(* Logix 5000 project; controller PRU vendor 1 type 14 code 107 rev 20.13; software revision 20.01; part 2 of 17 *)
(* tags used below, declared in another part *)
   RIGHT_ENCODER_DEG_OUT_REAL_OUT : REAL;
   LEFT_ENCODER_DEG_WAS_SCANRATE_MOVED_OUT : REAL;
   RIGHT_ENCODER_DEG_WAS_SCANRATE_MOVED_OUT : REAL;
   MASTER_RIGHT_BOOL_IN : BOOL;
   ENCODER_MOVED_LAST_SEC_REAL_OUT : REAL;
   MIX_REV_PER_MIN_REAL_OUT : REAL;
   RETENTION_TIME_MIN_REAL_OUT : REAL;
   MIX_FWD_PRESET_REAL_IN : REAL;
   MIX_REV_PRESET_REAL_IN : REAL;
   AUTO_FWD_CMD_BOOL_OUT : BOOL;
   ENCODER_ACC_REAL_OUT : REAL;
   SREW_MODE_INT_IN : INT;
   SCREW_PITCH_CONSTANT_REAL_IN : REAL;
   MIX_SEQ : INT;
   ONE_SECOND_ENCODER_SCAN : BOOL;   // 100 x 10mS.
   RIGHT_ENCODER_DEG_WAS_SCANRATE : REAL;
   MIX_SEQ_STEP_00_DONE_TON : TIMER;
   MIX_SEQ_STEP_01_DONE : BOOL;
   MIX_SEQ_STEP_02_DONE : BOOL;
   MIX_STEP_00_ION : BOOL;
   MIX_STEP_01_ION : BOOL;   // FORWARD
   MIX_STEP_01_ONSN : BOOL;
   MIX_STEP_01_ONSP : BOOL;
   MIX_FWD_SS : BOOL;
   MIX_CYC_TIME_ACC : DINT;
   MIX_CYC_TIME : REAL;
   MIX_FWD_DEG : REAL;
   MIX_DEG_PER_SEC : REAL;
   MIX_STEP_02_ION : BOOL;   // REVERSE
   FWD_CMD_BON : TIMER;
   REV_CMD_BON : TIMER;
   Revision : DINT;
   SCREW_ENCODERS : SCREW_ENCODERS;
   SCREW_SPEED : SCREW_SPEED;
(* SCREW_ENCODERS, continued *)

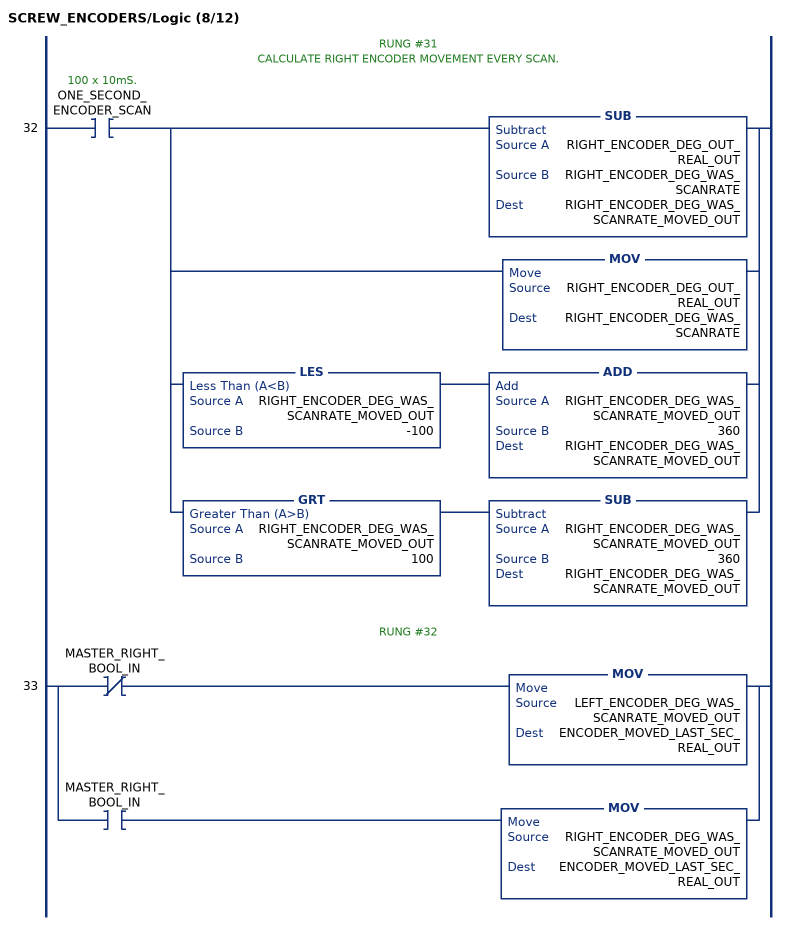
   // RUNG #31
   // CALCULATE RIGHT ENCODER MOVEMENT EVERY SCAN.
   32: XIC(ONE_SECOND_ENCODER_SCAN)[SUB(RIGHT_ENCODER_DEG_OUT_REAL_OUT,RIGHT_ENCODER_DEG_WAS_SCANRATE,RIGHT_ENCODER_DEG_WAS_SCANRATE_MOVED_OUT) ,MOV(RIGHT_ENCODER_DEG_OUT_REAL_OUT,RIGHT_ENCODER_DEG_WAS_SCANRATE) ,LES(RIGHT_ENCODER_DEG_WAS_SCANRATE_MOVED_OUT,-100) ADD(RIGHT_ENCODER_DEG_WAS_SCANRATE_MOVED_OUT,360,RIGHT_ENCODER_DEG_WAS_SCANRATE_MOVED_OUT) ,GRT(RIGHT_ENCODER_DEG_WAS_SCANRATE_MOVED_OUT,100) SUB(RIGHT_ENCODER_DEG_WAS_SCANRATE_MOVED_OUT,360,RIGHT_ENCODER_DEG_WAS_SCANRATE_MOVED_OUT) ];
   // RUNG #32
   33: [XIO(MASTER_RIGHT_BOOL_IN) MOV(LEFT_ENCODER_DEG_WAS_SCANRATE_MOVED_OUT,ENCODER_MOVED_LAST_SEC_REAL_OUT) ,XIC(MASTER_RIGHT_BOOL_IN) MOV(RIGHT_ENCODER_DEG_WAS_SCANRATE_MOVED_OUT,ENCODER_MOVED_LAST_SEC_REAL_OUT) ];
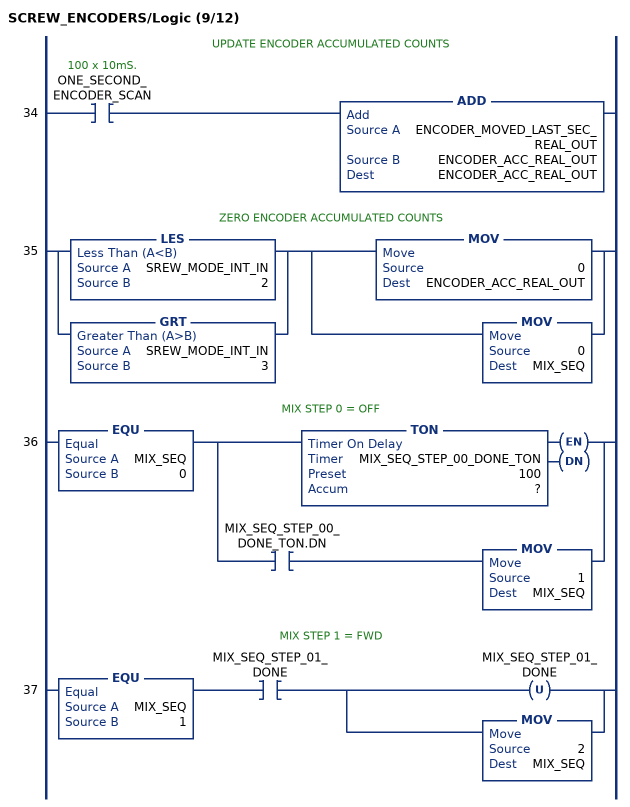
   // UPDATE ENCODER ACCUMULATED COUNTS
   34: XIC(ONE_SECOND_ENCODER_SCAN)ADD(ENCODER_MOVED_LAST_SEC_REAL_OUT,ENCODER_ACC_REAL_OUT,ENCODER_ACC_REAL_OUT);
   // ZERO ENCODER ACCUMULATED COUNTS
   35: [LES(SREW_MODE_INT_IN,2) ,GRT(SREW_MODE_INT_IN,3) ][MOV(0,ENCODER_ACC_REAL_OUT) ,MOV(0,MIX_SEQ) ];
   // MIX STEP 0 = OFF
   36: EQU(MIX_SEQ,0)[TON(MIX_SEQ_STEP_00_DONE_TON,?,?) ,XIC(MIX_SEQ_STEP_00_DONE_TON.DN) MOV(1,MIX_SEQ) ];
   // MIX STEP 1 = FWD
   37: EQU(MIX_SEQ,1)XIC(MIX_SEQ_STEP_01_DONE)[OTU(MIX_SEQ_STEP_01_DONE) ,MOV(2,MIX_SEQ) ];
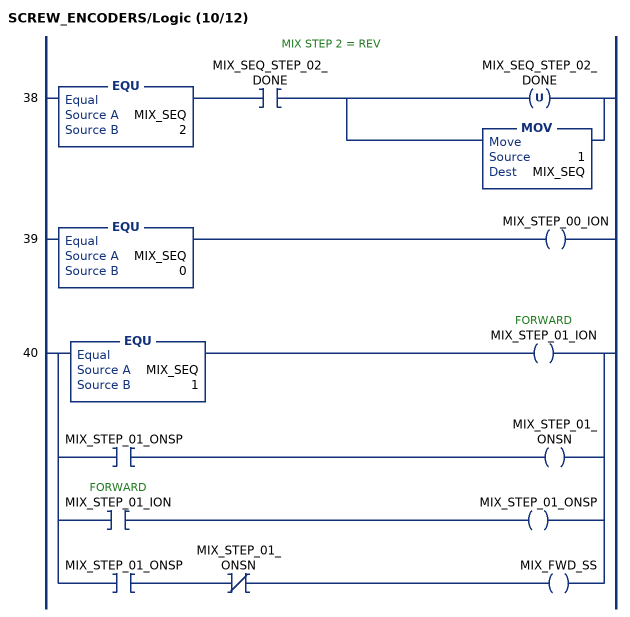
   // MIX STEP 2 = REV
   38: EQU(MIX_SEQ,2)XIC(MIX_SEQ_STEP_02_DONE)[OTU(MIX_SEQ_STEP_02_DONE) ,MOV(1,MIX_SEQ) ];
   39: EQU(MIX_SEQ,0)OTE(MIX_STEP_00_ION);
   40: [EQU(MIX_SEQ,1) OTE(MIX_STEP_01_ION) ,XIC(MIX_STEP_01_ONSP) OTE(MIX_STEP_01_ONSN) ,XIC(MIX_STEP_01_ION) OTE(MIX_STEP_01_ONSP) ,XIC(MIX_STEP_01_ONSP) XIO(MIX_STEP_01_ONSN) OTE(MIX_FWD_SS) ];
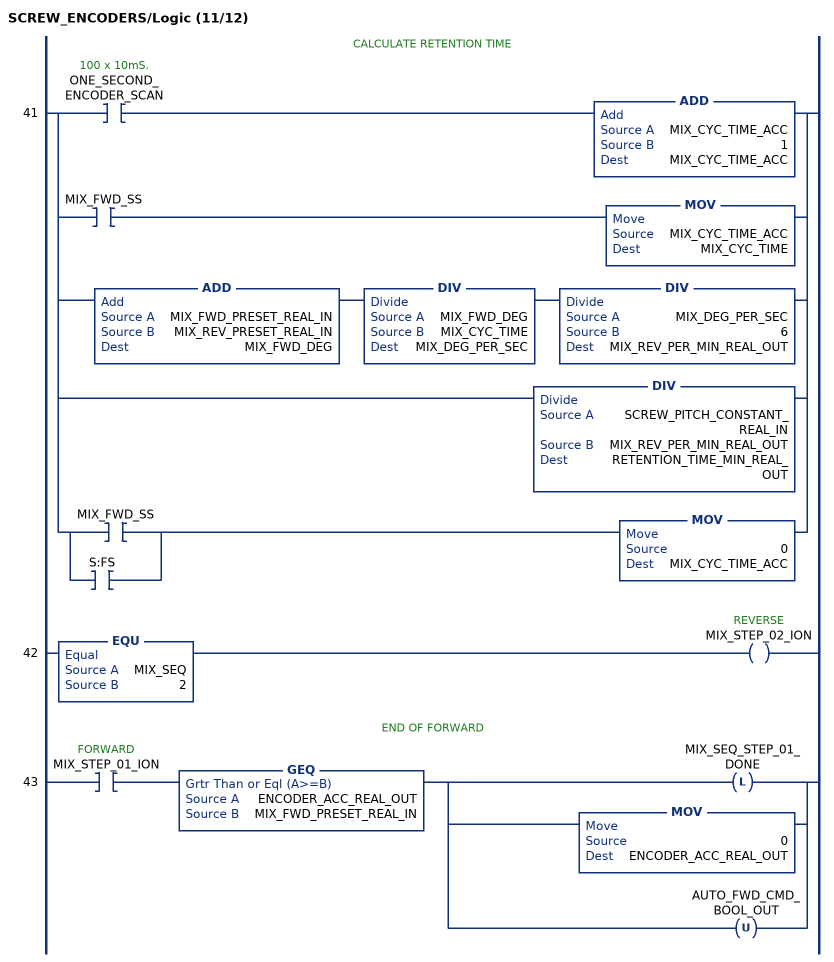
   // CALCULATE RETENTION TIME
   41: [XIC(ONE_SECOND_ENCODER_SCAN) ADD(MIX_CYC_TIME_ACC,1,MIX_CYC_TIME_ACC) ,XIC(MIX_FWD_SS) MOV(MIX_CYC_TIME_ACC,MIX_CYC_TIME) ,ADD(MIX_FWD_PRESET_REAL_IN,MIX_REV_PRESET_REAL_IN,MIX_FWD_DEG) DIV(MIX_FWD_DEG,MIX_CYC_TIME,MIX_DEG_PER_SEC) DIV(MIX_DEG_PER_SEC,6,MIX_REV_PER_MIN_REAL_OUT) ,DIV(SCREW_PITCH_CONSTANT_REAL_IN,MIX_REV_PER_MIN_REAL_OUT,RETENTION_TIME_MIN_REAL_OUT) ,[XIC(MIX_FWD_SS) ,XIC(S:FS) ] MOV(0,MIX_CYC_TIME_ACC) ];
   42: EQU(MIX_SEQ,2)OTE(MIX_STEP_02_ION);
   // END OF FORWARD
   43: XIC(MIX_STEP_01_ION)GEQ(ENCODER_ACC_REAL_OUT,MIX_FWD_PRESET_REAL_IN)[OTL(MIX_SEQ_STEP_01_DONE) ,MOV(0,ENCODER_ACC_REAL_OUT) ,OTU(AUTO_FWD_CMD_BOOL_OUT) ];
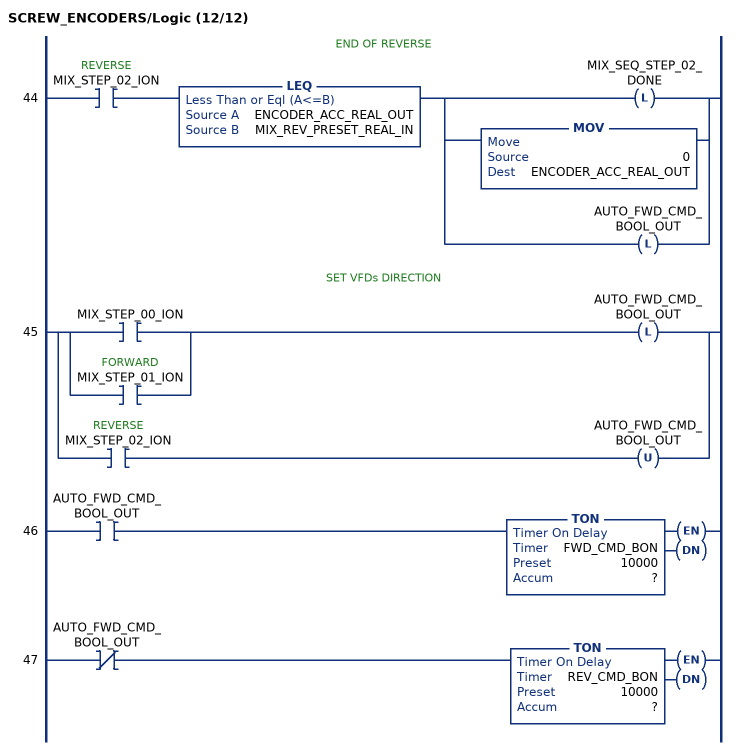
   // END OF REVERSE
   44: XIC(MIX_STEP_02_ION)LEQ(ENCODER_ACC_REAL_OUT,MIX_REV_PRESET_REAL_IN)[OTL(MIX_SEQ_STEP_02_DONE) ,MOV(0,ENCODER_ACC_REAL_OUT) ,OTL(AUTO_FWD_CMD_BOOL_OUT) ];
   // SET VFDs DIRECTION
   45: [[XIC(MIX_STEP_00_ION) ,XIC(MIX_STEP_01_ION) ] OTL(AUTO_FWD_CMD_BOOL_OUT) ,XIC(MIX_STEP_02_ION) OTU(AUTO_FWD_CMD_BOOL_OUT) ];
   46: XIC(AUTO_FWD_CMD_BOOL_OUT)TON(FWD_CMD_BON,?,?);
   47: XIO(AUTO_FWD_CMD_BOOL_OUT)TON(REV_CMD_BON,?,?);
END_ROUTINE
END_ADD_ON_INSTRUCTION

ADD_ON_INSTRUCTION SCREW_SPEED   (* revision 1.0, vendor Deterministic Systems, Inc. *)
VAR_INPUT
   IN_SCREW_MODE : INT; {required}
   IN_AUTO_FWD_CMD_BOOL : BOOL; {required}
   IN_MASTER_RIGHT_BOOL : BOOL; {required}
   IN_VFD_STOP_CMD : BOOL; {required}
   IN_DCS_AUTO_SCREW_CMD_PCNT : REAL; {required}
END_VAR
VAR_OUTPUT
   OUT_DCS_MASTER_SPEED_CMD : REAL; {access Read Only, required}
END_VAR
VAR_INPUT
   IN_HMI_SEMIAUTO_SCREW_CMD_PCNT : REAL; {required}
END_VAR
VAR_OUTPUT
   OUT_MASTER_AUTO_SETPOINT_PCNT : REAL; {access Read Only, required}
END_VAR
VAR_INPUT
   IN_LEFT_RIGHT_ENCODER_ERROR_DEG : REAL; {required}
   IN_WIPER_OSC_SETPOINT : REAL; {required}
END_VAR
VAR_OUTPUT
   OUT_FINAL_SCREW_POSITION_ERROR : REAL; {access Read Only, required}
   OUT_AUTO_SCREW_LEFT_CMD_FREQ : REAL; {access Read Only, required}
   OUT_AUTO_SCREW_RIGHT_CMD_FREQ : REAL; {access Read Only, required}
END_VAR
VAR_INPUT
   IN_LEFT_VFD_ION : BOOL; {required}
   IN_RIGHT_VFD_ION : BOOL; {required}
   IN_LEFT_VFD_ACTUAL : BOOL; {required}
   IN_RIGHT_VFD_ACTUAL : BOOL; {required}
END_VAR
VAR_OUTPUT
   OUT_FORCE_ZERO_SPEED : BOOL; {access Read Only, required}
END_VAR
VAR_INPUT
   IN_SCREW_FAULTED_IOK : BOOL; {required}
END_VAR
VAR_OUTPUT
   OUT_LEFT_AUTO_PCNT_SETPOINT : REAL; {access Read Only, required}
   OUT_RIGHT_AUTO_PCNT_SETPOINT : REAL; {access Read Only, required}
END_VAR
VAR_INPUT
   IN_LEFT_VFD_ACTUAL_FREQ : INT; {required}
   IN_RIGHT_VFD_ACTUAL_FREQ : INT; {required}
END_VAR
VAR_OUTPUT
   OUT_LEFT_VFD_ACTUAL_SPEED_PERCENT : REAL; {required}
   OUT_RIGHT_VFD_ACTUAL_SPEED_PERCENT : REAL; {access Read Only, required}
   CALC_COMP_LIMIT : REAL; {access None, required}
END_VAR
VAR_INPUT
   IN_SET_ZERO_SPEED : BOOL; {required}
END_VAR
VAR
   SCREW_MODE_AUTO : BOOL;
   DCS_MASTER_SPEED_CMD : REAL;
   SLAVE_COMPENSATION_GAIN : REAL;
   SLAVE_COMPENSATION_PER_DEGREE : REAL;
   SLAVE_AUTO_SETPOINT_PCNT : REAL;
   RIGHT_MAX_COMP_PCNT : REAL;
   RIGHT_MIN_COMP_PCNT : REAL;
   RPM_FREQ_MULTIPLIER : REAL := 711.16;
   MASTER_SETPOINT_END : REAL; {access None}
   CALC_MASTER_SETPOINT : REAL; {access None}
   ROC : DSi_COMP_SCALE; {access None}
   FWD_MASTER_AUTO_SETPOINT_PCNT : REAL; {access None}
   CALC_COMP_LIMIT_REV : REAL; {access None}
   REV_MASTER_AUTO_SETPOINT_PCNT : REAL; {access None}
   MASTER_SETPOINT_END_REV : REAL; {access None}
   ROC2 : DSi_COMP_SCALE; {access None}
END_VAR

ROUTINE Logic   (* ladder *)
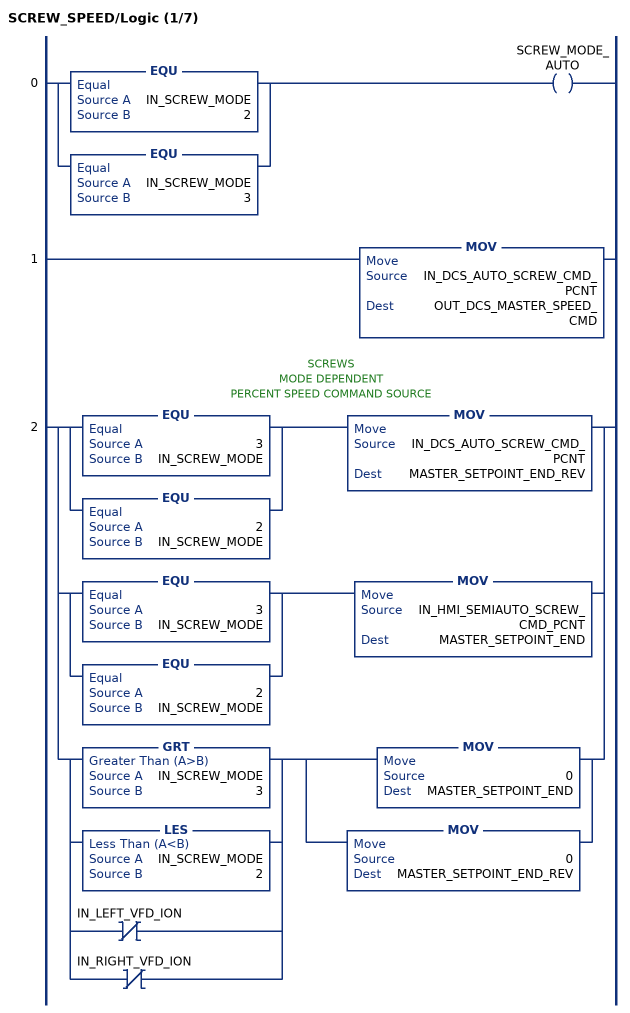
   0: [EQU(IN_SCREW_MODE,2) ,EQU(IN_SCREW_MODE,3) ]OTE(SCREW_MODE_AUTO);
   1: MOV(IN_DCS_AUTO_SCREW_CMD_PCNT,OUT_DCS_MASTER_SPEED_CMD);
   // SCREWS
   // MODE DEPENDENT
   // PERCENT SPEED COMMAND SOURCE
   2: [[EQU(3,IN_SCREW_MODE) ,EQU(2,IN_SCREW_MODE) ] MOV(IN_DCS_AUTO_SCREW_CMD_PCNT,MASTER_SETPOINT_END_REV) ,[EQU(3,IN_SCREW_MODE) ,EQU(2,IN_SCREW_MODE) ] MOV(IN_HMI_SEMIAUTO_SCREW_CMD_PCNT,MASTER_SETPOINT_END) ,[GRT(IN_SCREW_MODE,3) ,LES(IN_SCREW_MODE,2) ,XIO(IN_LEFT_VFD_ION) ,XIO(IN_RIGHT_VFD_ION) ] [MOV(0,MASTER_SETPOINT_END) ,MOV(0,MASTER_SETPOINT_END_REV) ] ];
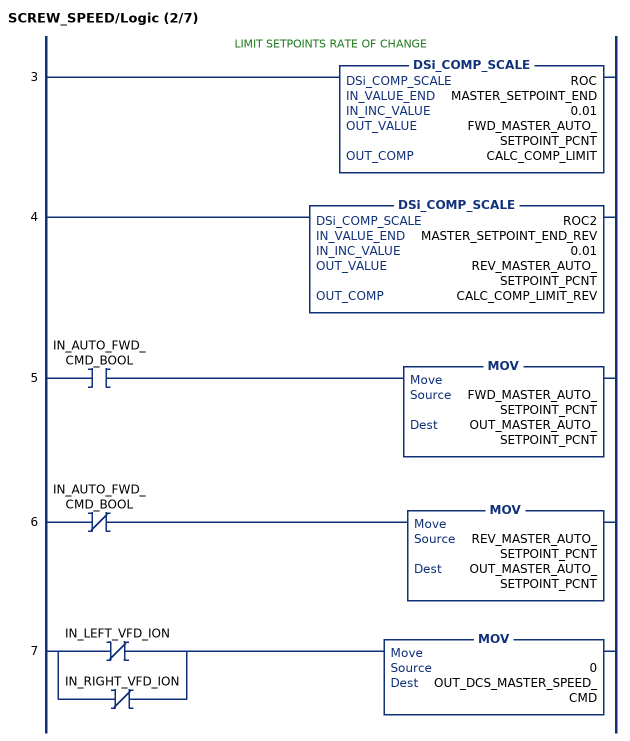
   // LIMIT SETPOINTS RATE OF CHANGE
   3: DSi_COMP_SCALE(ROC,MASTER_SETPOINT_END,0.01,FWD_MASTER_AUTO_SETPOINT_PCNT,CALC_COMP_LIMIT);
   4: DSi_COMP_SCALE(ROC2,MASTER_SETPOINT_END_REV,0.01,REV_MASTER_AUTO_SETPOINT_PCNT,CALC_COMP_LIMIT_REV);
   5: XIC(IN_AUTO_FWD_CMD_BOOL)MOV(FWD_MASTER_AUTO_SETPOINT_PCNT,OUT_MASTER_AUTO_SETPOINT_PCNT);
   6: XIO(IN_AUTO_FWD_CMD_BOOL)MOV(REV_MASTER_AUTO_SETPOINT_PCNT,OUT_MASTER_AUTO_SETPOINT_PCNT);
   7: [XIO(IN_LEFT_VFD_ION) ,XIO(IN_RIGHT_VFD_ION) ]MOV(0,OUT_DCS_MASTER_SPEED_CMD);
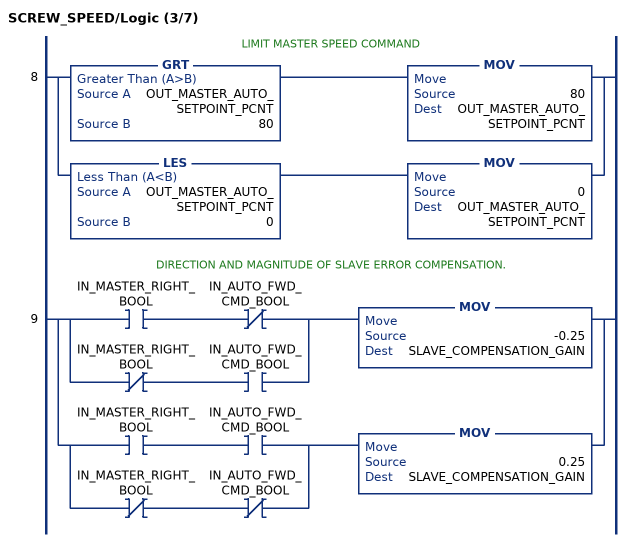
   // LIMIT MASTER SPEED COMMAND
   8: [GRT(OUT_MASTER_AUTO_SETPOINT_PCNT,80) MOV(80,OUT_MASTER_AUTO_SETPOINT_PCNT) ,LES(OUT_MASTER_AUTO_SETPOINT_PCNT,0) MOV(0,OUT_MASTER_AUTO_SETPOINT_PCNT) ];
   // DIRECTION AND MAGNITUDE OF SLAVE ERROR COMPENSATION.
   9: [[XIC(IN_MASTER_RIGHT_BOOL) XIO(IN_AUTO_FWD_CMD_BOOL) ,XIO(IN_MASTER_RIGHT_BOOL) XIC(IN_AUTO_FWD_CMD_BOOL) ] MOV(-0.25,SLAVE_COMPENSATION_GAIN) ,[XIC(IN_MASTER_RIGHT_BOOL) XIC(IN_AUTO_FWD_CMD_BOOL) ,XIO(IN_MASTER_RIGHT_BOOL) XIO(IN_AUTO_FWD_CMD_BOOL) ] MOV(0.25,SLAVE_COMPENSATION_GAIN) ];
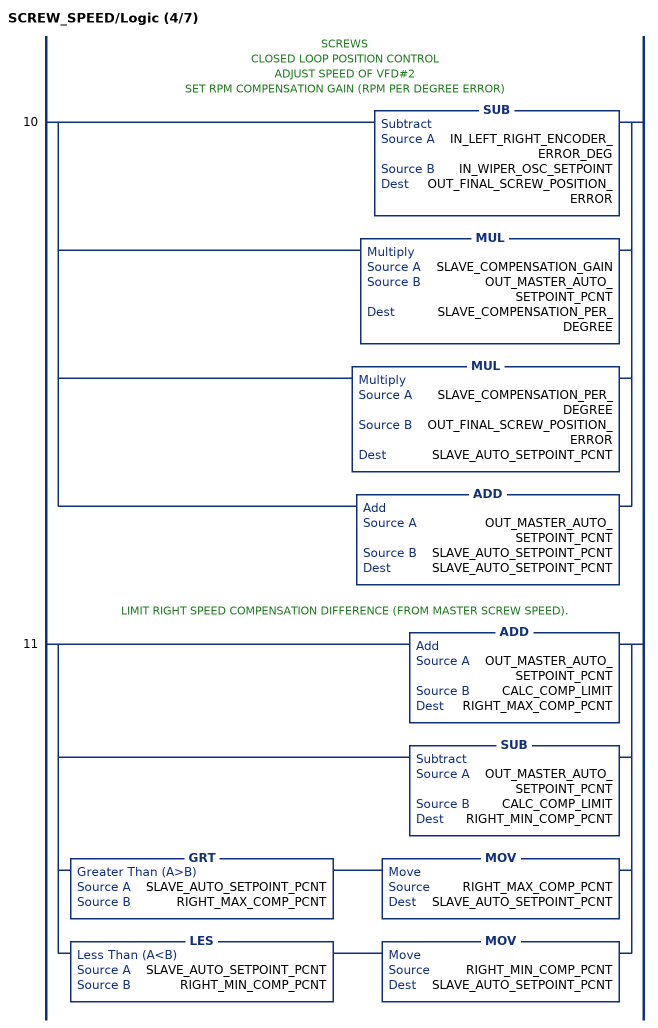
   // SCREWS
   // CLOSED LOOP POSITION CONTROL
   // ADJUST SPEED OF VFD#2
   // SET RPM COMPENSATION GAIN (RPM PER DEGREE ERROR)
   10: [SUB(IN_LEFT_RIGHT_ENCODER_ERROR_DEG,IN_WIPER_OSC_SETPOINT,OUT_FINAL_SCREW_POSITION_ERROR) ,MUL(SLAVE_COMPENSATION_GAIN,OUT_MASTER_AUTO_SETPOINT_PCNT,SLAVE_COMPENSATION_PER_DEGREE) ,MUL(SLAVE_COMPENSATION_PER_DEGREE,OUT_FINAL_SCREW_POSITION_ERROR,SLAVE_AUTO_SETPOINT_PCNT) ,ADD(OUT_MASTER_AUTO_SETPOINT_PCNT,SLAVE_AUTO_SETPOINT_PCNT,SLAVE_AUTO_SETPOINT_PCNT) ];
   // LIMIT RIGHT SPEED COMPENSATION DIFFERENCE (FROM MASTER SCREW SPEED).
   11: [ADD(OUT_MASTER_AUTO_SETPOINT_PCNT,CALC_COMP_LIMIT,RIGHT_MAX_COMP_PCNT) ,SUB(OUT_MASTER_AUTO_SETPOINT_PCNT,CALC_COMP_LIMIT,RIGHT_MIN_COMP_PCNT) ,GRT(SLAVE_AUTO_SETPOINT_PCNT,RIGHT_MAX_COMP_PCNT) MOV(RIGHT_MAX_COMP_PCNT,SLAVE_AUTO_SETPOINT_PCNT) ,LES(SLAVE_AUTO_SETPOINT_PCNT,RIGHT_MIN_COMP_PCNT) MOV(RIGHT_MIN_COMP_PCNT,SLAVE_AUTO_SETPOINT_PCNT) ];
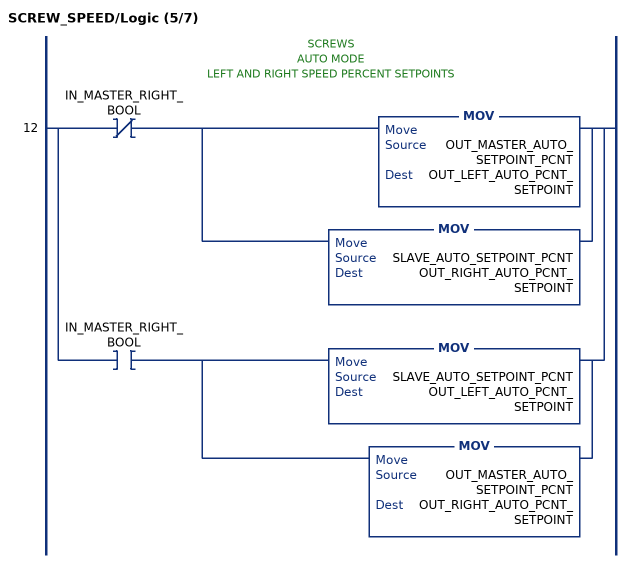
   // SCREWS
   // AUTO MODE
   // LEFT AND RIGHT SPEED PERCENT SETPOINTS
   12: [XIO(IN_MASTER_RIGHT_BOOL) [MOV(OUT_MASTER_AUTO_SETPOINT_PCNT,OUT_LEFT_AUTO_PCNT_SETPOINT) ,MOV(SLAVE_AUTO_SETPOINT_PCNT,OUT_RIGHT_AUTO_PCNT_SETPOINT) ] ,XIC(IN_MASTER_RIGHT_BOOL) [MOV(SLAVE_AUTO_SETPOINT_PCNT,OUT_LEFT_AUTO_PCNT_SETPOINT) ,MOV(OUT_MASTER_AUTO_SETPOINT_PCNT,OUT_RIGHT_AUTO_PCNT_SETPOINT) ] ];
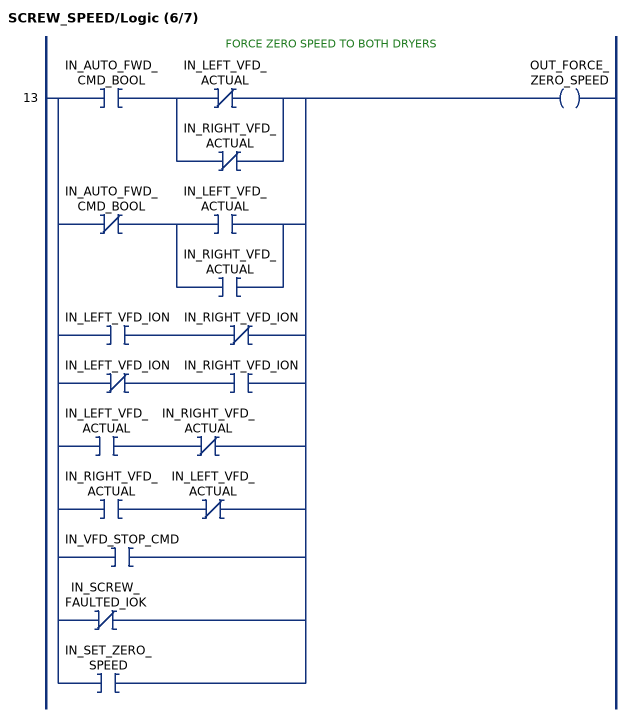
   // FORCE ZERO SPEED TO BOTH DRYERS
   13: [XIC(IN_AUTO_FWD_CMD_BOOL) [XIO(IN_LEFT_VFD_ACTUAL) ,XIO(IN_RIGHT_VFD_ACTUAL) ] ,XIO(IN_AUTO_FWD_CMD_BOOL) [XIC(IN_LEFT_VFD_ACTUAL) ,XIC(IN_RIGHT_VFD_ACTUAL) ] ,XIC(IN_LEFT_VFD_ION) XIO(IN_RIGHT_VFD_ION) ,XIO(IN_LEFT_VFD_ION) XIC(IN_RIGHT_VFD_ION) ,XIC(IN_LEFT_VFD_ACTUAL) XIO(IN_RIGHT_VFD_ACTUAL) ,XIC(IN_RIGHT_VFD_ACTUAL) XIO(IN_LEFT_VFD_ACTUAL) ,XIC(IN_VFD_STOP_CMD) ,XIO(IN_SCREW_FAULTED_IOK) ,XIC(IN_SET_ZERO_SPEED) ]OTE(OUT_FORCE_ZERO_SPEED);
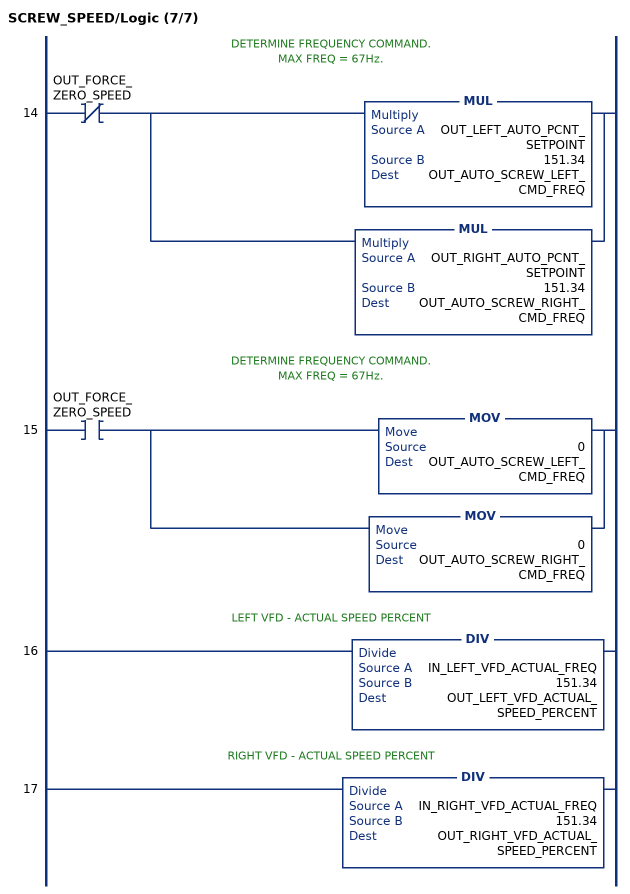
   // DETERMINE FREQUENCY COMMAND.
   // MAX FREQ = 67Hz.
   14: XIO(OUT_FORCE_ZERO_SPEED)[MUL(OUT_LEFT_AUTO_PCNT_SETPOINT,151.34,OUT_AUTO_SCREW_LEFT_CMD_FREQ) ,MUL(OUT_RIGHT_AUTO_PCNT_SETPOINT,151.34,OUT_AUTO_SCREW_RIGHT_CMD_FREQ) ];
   // DETERMINE FREQUENCY COMMAND.
   // MAX FREQ = 67Hz.
   15: XIC(OUT_FORCE_ZERO_SPEED)[MOV(0,OUT_AUTO_SCREW_LEFT_CMD_FREQ) ,MOV(0,OUT_AUTO_SCREW_RIGHT_CMD_FREQ) ];
   // LEFT VFD - ACTUAL SPEED PERCENT
   16: DIV(IN_LEFT_VFD_ACTUAL_FREQ,151.34,OUT_LEFT_VFD_ACTUAL_SPEED_PERCENT);
   // RIGHT VFD - ACTUAL SPEED PERCENT
   17: DIV(IN_RIGHT_VFD_ACTUAL_FREQ,151.34,OUT_RIGHT_VFD_ACTUAL_SPEED_PERCENT);
END_ROUTINE
END_ADD_ON_INSTRUCTION

ADD_ON_INSTRUCTION SCREW_WIPER   (* revision 1.0, vendor Deterministic Systems, Inc. *)
VAR_INPUT
   HMI_WIPE_INC_REAL_IN : REAL; {required}
   HMI_WIPE_SETPOINT_REAL_IN : REAL; {required}
   WIPE_HOLD_TIME_DINT_IN : DINT; {required}
END_VAR
VAR_OUTPUT
   WIPE_HOLDING_BOOL_OUT : BOOL; {access Read Only, required}
   WIPER_OSC_REAL_OUT : REAL; {access Read Only, required}
END_VAR
VAR_INPUT
   WIPE_EON_IN : BOOL; {required}
   WIPE_FREEZE_IN : BOOL; {required}
END_VAR
VAR
   SCREWS_TON : TIMER := (PRE := 10000);
   WIPE_INC : REAL;
   WIPE_PLUS_HOLD_VALUE : REAL;
   WIPE_MINUS_HOLD_VALUE : REAL;
   SCREWS_PLUS_HOLD_ONSN : BOOL;
   SCREWS_PLUS_HOLD_ONSP : BOOL;
   SCREWS_PLUS_HOLD_SS : BOOL;
   SCREWS_PLUS_HOLD : BOOL;
   SCREWS_MINUS_HOLD_ONSN : BOOL;
   SCREWS_MINUS_HOLD_ONSP : BOOL;
   SCREWS_MINUS_HOLD_SS : BOOL;
   SCREWS_MINUS_HOLD : BOOL;
   WIPE_HOLD_TIMER : TIMER := (PRE := 5000);
   WIPE_SIN_INDEX : REAL;
   WIPE_SINE : REAL;
   HMI_WIPE_SETPOINT_REAL : REAL; {access None}
   HMI_WIPE_SETPOINT_COMP : REAL; {access None}
   ROC_WIPE_SETPOINT : DSi_COMP_SCALE; {access None}
END_VAR

ROUTINE Logic   (* ladder *)
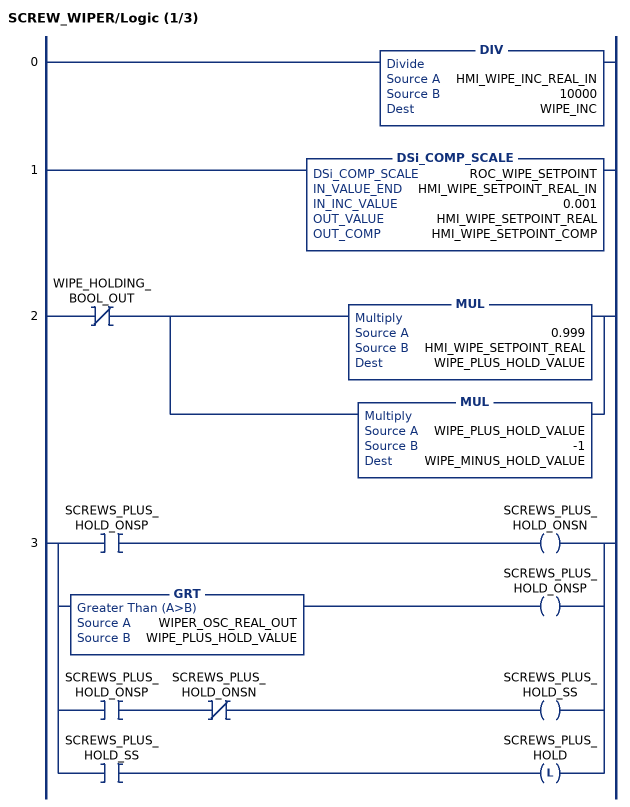
   0: DIV(HMI_WIPE_INC_REAL_IN,10000,WIPE_INC);
   1: DSi_COMP_SCALE(ROC_WIPE_SETPOINT,HMI_WIPE_SETPOINT_REAL_IN,0.001,HMI_WIPE_SETPOINT_REAL,HMI_WIPE_SETPOINT_COMP);
   2: XIO(WIPE_HOLDING_BOOL_OUT)[MUL(0.999,HMI_WIPE_SETPOINT_REAL,WIPE_PLUS_HOLD_VALUE) ,MUL(WIPE_PLUS_HOLD_VALUE,-1,WIPE_MINUS_HOLD_VALUE) ];
   3: [XIC(SCREWS_PLUS_HOLD_ONSP) OTE(SCREWS_PLUS_HOLD_ONSN) ,GRT(WIPER_OSC_REAL_OUT,WIPE_PLUS_HOLD_VALUE) OTE(SCREWS_PLUS_HOLD_ONSP) ,XIC(SCREWS_PLUS_HOLD_ONSP) XIO(SCREWS_PLUS_HOLD_ONSN) OTE(SCREWS_PLUS_HOLD_SS) ,XIC(SCREWS_PLUS_HOLD_SS) OTL(SCREWS_PLUS_HOLD) ];
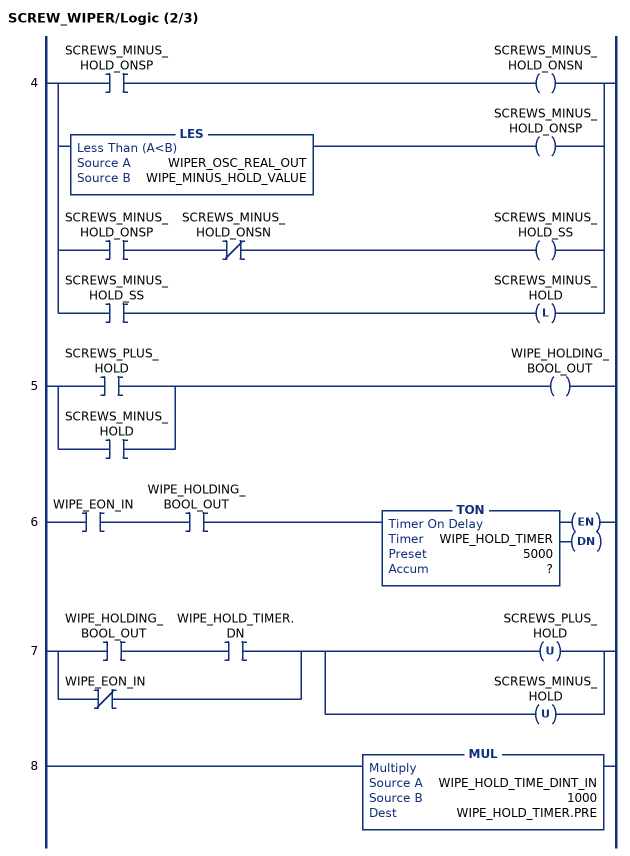
   4: [XIC(SCREWS_MINUS_HOLD_ONSP) OTE(SCREWS_MINUS_HOLD_ONSN) ,LES(WIPER_OSC_REAL_OUT,WIPE_MINUS_HOLD_VALUE) OTE(SCREWS_MINUS_HOLD_ONSP) ,XIC(SCREWS_MINUS_HOLD_ONSP) XIO(SCREWS_MINUS_HOLD_ONSN) OTE(SCREWS_MINUS_HOLD_SS) ,XIC(SCREWS_MINUS_HOLD_SS) OTL(SCREWS_MINUS_HOLD) ];
   5: [XIC(SCREWS_PLUS_HOLD) ,XIC(SCREWS_MINUS_HOLD) ]OTE(WIPE_HOLDING_BOOL_OUT);
   6: XIC(WIPE_EON_IN)XIC(WIPE_HOLDING_BOOL_OUT)TON(WIPE_HOLD_TIMER,?,?);
   7: [XIC(WIPE_HOLDING_BOOL_OUT) XIC(WIPE_HOLD_TIMER.DN) ,XIO(WIPE_EON_IN) ][OTU(SCREWS_PLUS_HOLD) ,OTU(SCREWS_MINUS_HOLD) ];
   8: MUL(WIPE_HOLD_TIME_DINT_IN,1000,WIPE_HOLD_TIMER.PRE);
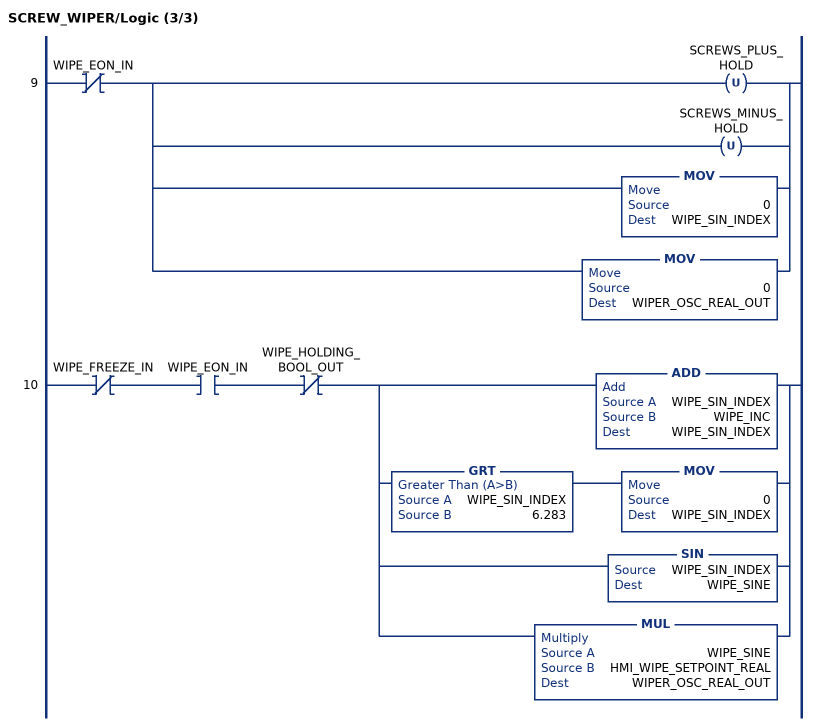
   9: XIO(WIPE_EON_IN)[OTU(SCREWS_PLUS_HOLD) ,OTU(SCREWS_MINUS_HOLD) ,MOV(0,WIPE_SIN_INDEX) ,MOV(0,WIPER_OSC_REAL_OUT) ];
   10: XIO(WIPE_FREEZE_IN)XIC(WIPE_EON_IN)XIO(WIPE_HOLDING_BOOL_OUT)[ADD(WIPE_SIN_INDEX,WIPE_INC,WIPE_SIN_INDEX) ,GRT(WIPE_SIN_INDEX,6.283) MOV(0,WIPE_SIN_INDEX) ,SIN(WIPE_SIN_INDEX,WIPE_SINE) ,MUL(WIPE_SINE,HMI_WIPE_SETPOINT_REAL,WIPER_OSC_REAL_OUT) ];
END_ROUTINE
END_ADD_ON_INSTRUCTION

ADD_ON_INSTRUCTION TE_SELECTED_AVE   (* revision 1.0, vendor Deterministic Systems, Inc. *)
VAR_INPUT
   IN_SEL_1ST_TE : BOOL; {required}
   IN_SEL_2ND_TE : BOOL; {required}
   IN_SEL_3RD_TE : BOOL; {required}
   IN_SEL_4TH_TE : BOOL; {required}
   IN_1ST_TE : REAL; {required}
   IN_2ND_TE : REAL; {required}
   IN_3RD_TE : REAL; {required}
   IN_4TH_TE : REAL; {required}
END_VAR
VAR_OUTPUT
   OUT_ZONE_1_AVE : REAL; {access Read Only, required}
END_VAR
VAR
   ZONE_1_TEMP_TOTAL : REAL; {access None}
   ZONE_1_TEMP_SEL_NUM : REAL; {access None}
   TEMP_ZONE_1_AVE : REAL; {access None}
END_VAR

ROUTINE Logic   (* ladder *)
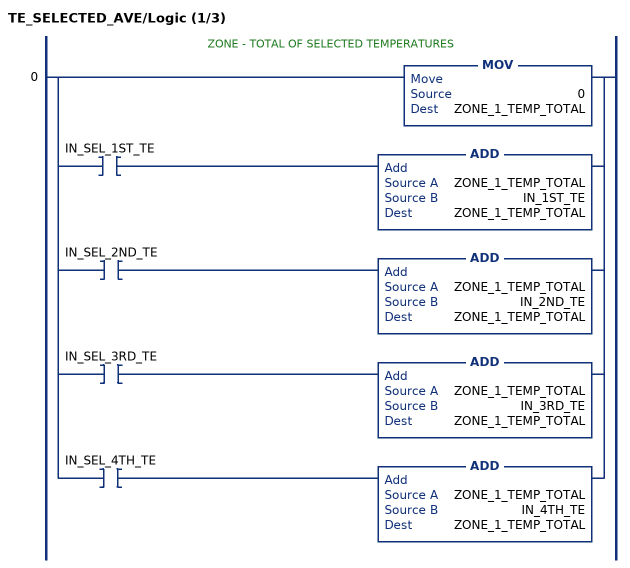
   // ZONE - TOTAL OF SELECTED TEMPERATURES
   0: [MOV(0,ZONE_1_TEMP_TOTAL) ,XIC(IN_SEL_1ST_TE) ADD(ZONE_1_TEMP_TOTAL,IN_1ST_TE,ZONE_1_TEMP_TOTAL) ,XIC(IN_SEL_2ND_TE) ADD(ZONE_1_TEMP_TOTAL,IN_2ND_TE,ZONE_1_TEMP_TOTAL) ,XIC(IN_SEL_3RD_TE) ADD(ZONE_1_TEMP_TOTAL,IN_3RD_TE,ZONE_1_TEMP_TOTAL) ,XIC(IN_SEL_4TH_TE) ADD(ZONE_1_TEMP_TOTAL,IN_4TH_TE,ZONE_1_TEMP_TOTAL) ];
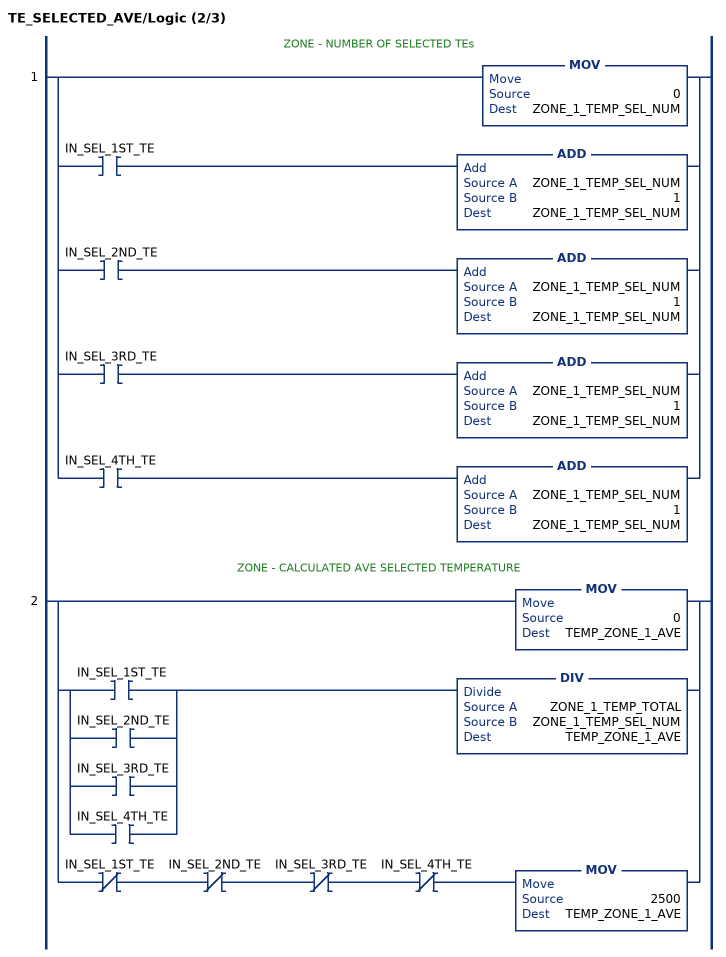
   // ZONE - NUMBER OF SELECTED TEs
   1: [MOV(0,ZONE_1_TEMP_SEL_NUM) ,XIC(IN_SEL_1ST_TE) ADD(ZONE_1_TEMP_SEL_NUM,1,ZONE_1_TEMP_SEL_NUM) ,XIC(IN_SEL_2ND_TE) ADD(ZONE_1_TEMP_SEL_NUM,1,ZONE_1_TEMP_SEL_NUM) ,XIC(IN_SEL_3RD_TE) ADD(ZONE_1_TEMP_SEL_NUM,1,ZONE_1_TEMP_SEL_NUM) ,XIC(IN_SEL_4TH_TE) ADD(ZONE_1_TEMP_SEL_NUM,1,ZONE_1_TEMP_SEL_NUM) ];
   // ZONE - CALCULATED AVE SELECTED TEMPERATURE
   2: [MOV(0,TEMP_ZONE_1_AVE) ,[XIC(IN_SEL_1ST_TE) ,XIC(IN_SEL_2ND_TE) ,XIC(IN_SEL_3RD_TE) ,XIC(IN_SEL_4TH_TE) ] DIV(ZONE_1_TEMP_TOTAL,ZONE_1_TEMP_SEL_NUM,TEMP_ZONE_1_AVE) ,XIO(IN_SEL_1ST_TE) XIO(IN_SEL_2ND_TE) XIO(IN_SEL_3RD_TE) XIO(IN_SEL_4TH_TE) MOV(2500,TEMP_ZONE_1_AVE) ];
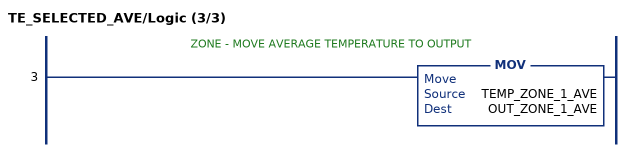
   // ZONE - MOVE AVERAGE TEMPERATURE TO OUTPUT
   3: MOV(TEMP_ZONE_1_AVE,OUT_ZONE_1_AVE);
END_ROUTINE
END_ADD_ON_INSTRUCTION
